FUNCTION_BLOCK FieldsToArrowheadService (* Translate individual fields to an ArrowheadService type *)
  (* Standard: 61499-2; Description: Copyright (c) 2018 fortiss GmbH This program and the accompanying materials are made available under the terms of the Eclipse Public License 2.0 which is available at https://www.eclipse.org/legal/epl-2.0/ SPDX-License-Identifier: EPL-2.0 *)
  (* Version 1.0, 2018-09-21, Jose Cabral, fortiss GmbH *)
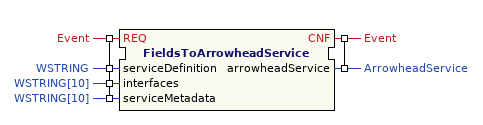
  EVENT_INPUT
    REQ WITH serviceDefinition, interfaces, serviceMetadata; (* Create arrowhead service *)
  END_EVENT
  EVENT_OUTPUT
    CNF WITH arrowheadService; (* Arrowhead service created *)
  END_EVENT
  VAR_INPUT
    serviceDefinition : WSTRING; (* Identification of the service *)
    interfaces : ARRAY [0..9] OF WSTRING; (* Interfaces implemented by the service *)
    serviceMetadata : ARRAY [0..9] OF WSTRING; (* Metadata of the service in key=value format *)
  END_VAR
  VAR_OUTPUT
    arrowheadService : ArrowheadService; (* Created Arrowhead service *)
  END_VAR
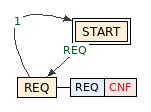
  EC_STATES
    START; (* Initial State *)
    REQ : REQ -> CNF; (* Normal execution *)
  END_STATES
  EC_TRANSITIONS
    START TO REQ := REQ;
    REQ TO START := 1;
  END_TRANSITIONS
  ALGORITHM REQ IN ST:
VAR_TEMP
	i : INT;
END_VAR
;

i := 0;
arrowheadService.serviceDefinition := serviceDefinition;

WHILE i < 10 DO // looks like while is faster than FOR when exporting to cpp
	arrowheadService.interfaces[i] := interfaces[i];
	arrowheadService.serviceMetadata[i] := serviceMetadata[i];
	i := i + 1;
END_WHILE;
  END_ALGORITHM
END_FUNCTION_BLOCK
